// TIA Portal V19 export
TYPE "typeU3Em1Para"
// stored: Access Published
   STRUCT
      cm1AxisControl : "typeAxisControlInterface";
      cm12 { S7_SetPoint := 'True'} : "LAF_typeNgStrapParameters";
   END_STRUCT;
END_TYPE
